FUNCTION F_LminToSI : LREAL
VAR_INPUT
	fLmin : LREAL;
END_VAR
VAR
END_VAR

F_LminToSI := fLmin / 60000;

END_FUNCTION

(* stored: Version 1.1.0.1, ProductVersion 3.1.4024.10
   POU F_LminToSI: Id {94d741d9-9c67-46ea-969d-523fa1c7f352}, SpecialFunc None *)
